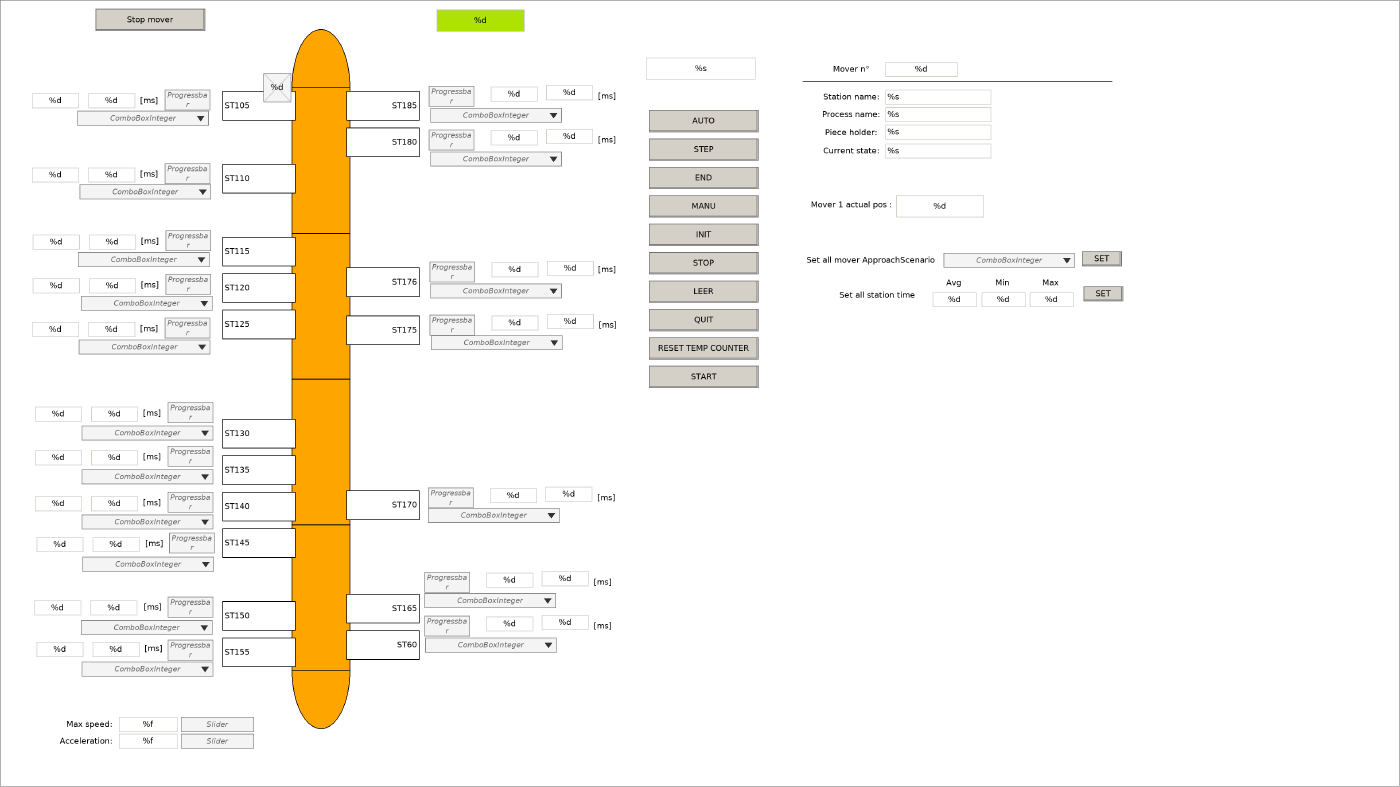
VISUALIZATION VISU_main  // 1920x1080
    Ellipse (400,840 80x160)
    Rectangle (400,720 80x200)
    Rectangle (400,520 80x200)
    Rectangle (400,320 80x200)
    Ellipse (400,40 80x160)
    Rectangle (400,120 80x200)
    Button (890,151 150x30), "AUTO", colour toggle: HMI.btArMain[0].on, input disabled if: HMI.btArMain[0].disable
        tap HMI.btArMain[0].button
    Button (890,190 150x30), "STEP", colour toggle: HMI.btArMain[1].on, input disabled if: HMI.btArMain[1].disable
        tap HMI.btArMain[1].button
    Button (890,229 150x30), "END", colour toggle: HMI.btArMain[2].on, input disabled if: HMI.btArMain[2].disable
        tap HMI.btArMain[2].button
    Button (890,307 150x30), "INIT", colour toggle: HMI.btArMain[4].on, input disabled if: HMI.btArMain[4].disable
        tap HMI.btArMain[4].button
    Button (890,346 150x30), "STOP", colour toggle: HMI.btArMain[5].disable, input disabled if: HMI.btArMain[5].disable
        tap HMI.btArMain[5].button
    Button (890,385 150x30), "LEER", colour toggle: HMI.btArMain[6].disable, input disabled if: HMI.btArMain[6].disable
        tap HMI.btArMain[6].button
    Button (890,424 150x30), "QUIT", colour toggle: HMI.btArMain[7].disable, input disabled if: HMI.btArMain[7].disable
        tap HMI.btArMain[7].button
    Button (890,463 150x30), "RESET TEMP COUNTER", colour toggle: HMI.btArMain[8].disable, input disabled if: HMI.btArMain[8].disable
        tap HMI.btArMain[8].button
    Button (890,268 150x30), "MANU", colour toggle: HMI.btArMain[3].on, input disabled if: HMI.btArMain[3].disable
        tap HMI.btArMain[3].button
    Textfield (886,79 150x30), "%s", text variable: _14_STATE.sStateDbg
    Button (890,502 150x30), "START", colour toggle: HMI.btArMain[9].disable, input disabled if: HMI.btArMain[9].disable
        tap HMI.btArMain[9].button
    Rectangle (475,175 100x40), "ST180", colour toggle: NOT PRG.st180_aut.xMoverPathFree
    Rectangle (475,367 100x40), "ST176", colour toggle: NOT PRG.st176_aut.xMoverPathFree
    Rectangle (475,433 100x40), "ST175", colour toggle: NOT PRG.st170_aut.xMoverPathFree
    Rectangle (475,673 100x40), "ST170", colour toggle: NOT PRG.st170_aut.xMoverPathFree
    Rectangle (475,815 100x40), "ST165", colour toggle: NOT PRG.st165_aut.xMoverPathFree
    Rectangle (475,865 100x40), "ST60", colour toggle: NOT PRG.st160_aut.xMoverPathFree
    Rectangle (305,875 100x40), "ST155", colour toggle: NOT PRG.st155_aut.xMoverPathFree
    Rectangle (475,125 100x40), "ST185", colour toggle: NOT PRG.st185_aut.xMoverPathFree
    Progressbar (588,178 62x28), variable: SIMU.iCompletionHMI[17]
    Progressbar (589,359 62x28), variable: SIMU.iCompletionHMI[16]
    Progressbar (589,432 62x28), variable: SIMU.iCompletionHMI[15]
    Progressbar (587,669 62x28), variable: SIMU.iCompletionHMI[14]
    Progressbar (582,785 62x28), variable: SIMU.iCompletionHMI[13]
    Progressbar (582,845 62x28), variable: SIMU.iCompletionHMI[12]
    Progressbar (230,878 62x28), variable: SIMU.iCompletionHMI[11]
    Progressbar (588,118 62x28), variable: SIMU.iCompletionHMI[18]
    Textfield (749,177 64x20), "%d", text variable: PERS.iStationTimeDef2[17]
        OnMouseDown: write the text variable via Default
    Label (805,177 55x30), "[ms]"
    Textfield (750,358 64x20), "%d", text variable: PERS.iStationTimeDef2[16]
        OnMouseDown: write the text variable via Default
    Label (805,355 55x30), "[ms]"
    Textfield (750,431 64x20), "%d", text variable: PERS.iStationTimeDef2[15]
        OnMouseDown: write the text variable via Default
    Label (806,431 55x30), "[ms]"
    Textfield (748,668 64x20), "%d", text variable: PERS.iStationTimeDef2[14]
        OnMouseDown: write the text variable via Default
    Label (804,668 55x30), "[ms]"
    Textfield (743,784 64x20), "%d", text variable: PERS.iStationTimeDef2[13]
        OnMouseDown: write the text variable via Default
    Label (799,784 55x30), "[ms]"
    Textfield (743,844 64x20), "%d", text variable: PERS.iStationTimeDef2[12]
        OnMouseDown: write the text variable via Default
    Label (799,844 55x30), "[ms]"
    Textfield (127,881 64x20), "%d", text variable: PERS.iStationTimeDef2[11]
        OnMouseDown: write the text variable via Default
    Label (183,875 55x30), "[ms]"
    Textfield (749,117 64x20), "%d", text variable: PERS.iStationTimeDef2[18]
        OnMouseDown: write the text variable via Default
    Label (805,117 55x30), "[ms]"
    Textfield (1229,268 120x30), "%d", text variable: MAIN.MoverMan._MoverList[1]._MoverAxis._CurrentPos
        OnMouseDown: write the text variable via Default
    Label (1080,266 146x30), "Mover 1 actual pos :"
    Textfield (599,13 120x30), "%d", text variable: PERS.iRecipeCurrent
        OnMouseDown: write the text variable via Default
    ComboBoxInteger (590,148 180x20), variable: MAIN.MoverMan._StationList[18]._ApproachScenario
    ComboBoxInteger (590,208 180x20), variable: MAIN.MoverMan._StationList[17]._ApproachScenario
    ComboBoxInteger (590,389 180x20), variable: MAIN.MoverMan._StationList[16]._ApproachScenario
    ComboBoxInteger (591,460 180x20), variable: MAIN.MoverMan._StationList[15]._ApproachScenario
    ComboBoxInteger (587,697 180x20), variable: MAIN.MoverMan._StationList[14]._ApproachScenario
    ComboBoxInteger (582,814 180x20), variable: MAIN.MoverMan._StationList[13]._ApproachScenario
    ComboBoxInteger (583,875 180x20), variable: MAIN.MoverMan._StationList[12]._ApproachScenario
    ComboBoxInteger (112,908 180x20), variable: MAIN.MoverMan._StationList[11]._ApproachScenario
    Rectangle (305,825 100x40), "ST150", colour toggle: NOT PRG.st150_aut.xMoverPathFree
    Progressbar (230,819 62x28), variable: SIMU.iCompletionHMI[10]
    Textfield (124,824 64x20), "%d", text variable: PERS.iStationTimeDef2[10]
        OnMouseDown: write the text variable via Default
    Label (182,818 55x30), "[ms]"
    ComboBoxInteger (111,851 180x20), variable: MAIN.MoverMan._StationList[10]._ApproachScenario
    Textfield (127,737 64x20), "%d", text variable: PERS.iStationTimeDef2[9]
        OnMouseDown: write the text variable via Default
    Label (184,731 55x30), "[ms]"
    Rectangle (305,725 100x40), "ST145", colour toggle: NOT PRG.st105_aut.xMoverPathFree
    Progressbar (232,731 62x28), variable: SIMU.iCompletionHMI[9]
    ComboBoxInteger (113,764 180x20), variable: MAIN.MoverMan._StationList[9]._ApproachScenario
    Textfield (125,681 64x20), "%d", text variable: PERS.iStationTimeDef2[8]
        OnMouseDown: write the text variable via Default
    Label (181,675 55x30), "[ms]"
    Rectangle (305,675 100x40), "ST140", colour toggle: NOT PRG.st140_aut.xMoverPathFree
    Progressbar (230,675 62x28), variable: SIMU.iCompletionHMI[8]
    ComboBoxInteger (112,706 180x20), variable: MAIN.MoverMan._StationList[8]._ApproachScenario
    Textfield (125,618 64x20), "%d", text variable: PERS.iStationTimeDef2[7]
        OnMouseDown: write the text variable via Default
    Label (181,612 55x30), "[ms]"
    Rectangle (305,625 100x40), "ST135", colour toggle: NOT PRG.st135_aut.xMoverPathFree
    Progressbar (230,612 62x28), variable: SIMU.iCompletionHMI[7]
    ComboBoxInteger (112,644 180x20), variable: MAIN.MoverMan._StationList[7]._ApproachScenario
    Textfield (125,558 64x20), "%d", text variable: PERS.iStationTimeDef2[6]
        OnMouseDown: write the text variable via Default
    Label (181,552 55x30), "[ms]"
    Rectangle (305,575 100x40), "ST130", colour toggle: NOT PRG.st130_aut.xMoverPathFree
    Progressbar (230,552 62x28), variable: SIMU.iCompletionHMI[6]
    ComboBoxInteger (112,584 180x20), variable: MAIN.MoverMan._StationList[6]._ApproachScenario
    Textfield (121,442 64x20), "%d", text variable: PERS.iStationTimeDef2[5]
        OnMouseDown: write the text variable via Default
    Label (177,436 55x30), "[ms]"
    Rectangle (305,425 100x40), "ST125", colour toggle: NOT PRG.st125_aut.xMoverPathFree
    Progressbar (226,436 62x28), variable: SIMU.iCompletionHMI[5]
    ComboBoxInteger (108,466 180x20), variable: MAIN.MoverMan._StationList[5]._ApproachScenario
    Textfield (122,382 64x20), "%d", text variable: PERS.iStationTimeDef2[4]
        OnMouseDown: write the text variable via Default
    Label (178,376 55x30), "[ms]"
    Rectangle (305,375 100x40), "ST120", colour toggle: NOT PRG.st120_aut.xMoverPathFree
    Progressbar (227,376 62x28), variable: SIMU.iCompletionHMI[4]
    ComboBoxInteger (111,406 180x20), variable: MAIN.MoverMan._StationList[4]._ApproachScenario
    Textfield (122,322 64x20), "%d", text variable: PERS.iStationTimeDef2[3]
        OnMouseDown: write the text variable via Default
    Label (178,316 55x30), "[ms]"
    Rectangle (305,325 100x40), "ST115", colour toggle: NOT PRG.st115_aut.xMoverPathFree
    Progressbar (227,316 62x28), variable: SIMU.iCompletionHMI[3]
    ComboBoxInteger (107,346 180x20), variable: MAIN.MoverMan._StationList[3]._ApproachScenario
    Textfield (121,230 64x20), "%d", text variable: PERS.iStationTimeDef2[2]
        OnMouseDown: write the text variable via Default
    Label (177,224 55x30), "[ms]"
    Rectangle (305,225 100x40), "ST110", colour toggle: NOT PRG.st110_aut.xMoverPathFree
    Progressbar (226,224 62x28), variable: SIMU.iCompletionHMI[2]
    ComboBoxInteger (109,253 180x20), variable: MAIN.MoverMan._StationList[2]._ApproachScenario
    Rectangle (305,125 100x40), "ST105", colour toggle: NOT PRG.st105_aut.xMoverPathFree
    Progressbar (226,123 62x28), variable: SIMU.iCompletionHMI[1]
    Textfield (121,128 64x20), "%d", text variable: PERS.iStationTimeDef2[1]
        OnMouseDown: write the text variable via Edit
    Label (177,123 55x30), "[ms]"
    ComboBoxInteger (106,152 180x20), variable: MAIN.MoverMan._StationList[1]._ApproachScenario
    ComboBoxInteger (1294,347 180x20), variable: MAIN.MoverMan.HMI_Scenario
    Label (1098,342 187x30), "Set all mover ApproachScenario"
    Button (1484,345 54x20), "SET"
        OnMouseDown: execute { MAIN.MoverMan.SetAllScenario(); }
    Label (1132,390 126x30), "Set all station time"
    Textfield (1279,401 60x20), "%d", text variable: MAIN.MoverMan.HMI_TimeAvg
        OnMouseDown: write the text variable via Default
    Label (1280,377 56x22), "Avg"
    Textfield (1346,401 60x20), "%d", text variable: MAIN.MoverMan.HMI_TimeMin
        OnMouseDown: write the text variable via Default
    Label (1347,377 56x22), "Min"
    Textfield (1412,401 60x20), "%d", text variable: MAIN.MoverMan.HMI_TimeMax
        OnMouseDown: write the text variable via Default
    Label (1413,377 56x22), "Max"
    Button (1486,393 54x20), "SET"
        OnMouseDown: execute { MAIN.MoverMan.SetAllTimers(ADR(PERS.iStationTimeDef1), 0); MAIN.MoverMan.SetAllTimers(ADR(PERS.iStationTimeDef2), 500); }
    Button (131,12 150x30), "Stop mover", colour toggle: MAIN.MoverMan.HMI_xStopMover
        toggle MAIN.MoverMan.HMI_xStopMover
    Label (1118,80 99x30), "Mover n°"
    Line (1101,111) (1525,111)
    Label (1118,118 99x30), "Station name:"
    Label (1118,142 99x30), "Process name:"
    Label (1118,167 99x30), "Piece holder:"
    Label (1118,192 99x30), "Current state:"
    Textfield (1214,85 99x20), "%d", text variable: MAIN.MoverMan.HMI_iSelMover
        OnMouseDown: write the text variable via Default
    Textfield (1214,123 145x20), "%s", text variable: MAIN.MoverMan._MoverList[MAIN.MoverMan.HMI_iSelMover].Station.ToString()
    Textfield (1214,147 145x20), "%s", text variable: MAIN.MoverMan._MoverList[MAIN.MoverMan.HMI_iSelMover].Station.Process.ToString()
    Textfield (1214,171 145x20), "%s"
    Textfield (1214,197 145x20), "%s", text variable: TO_STRING(MAIN.MoverMan._MoverList[MAIN.MoverMan.HMI_iSelMover]._State)
    Image (361,100 38x40), "%d", text variable: MAIN.MoverMan._MoverList[1]._ID, colour toggle: MAIN.MoverMan._SimuMoverList[1]._xStuck, invisible if: MAIN.MoverMan._MoverList[1]._MoverAxis._iID>CONST.MOVER_NUMBER, image: Custom.MoverSimu_final
        p3560616238: MAIN.MoverMan._MoverList[1]._MoverAxis.outSimuCurrentPos.x
        p2738717112: MAIN.MoverMan._MoverList[1]._MoverAxis.outSimuCurrentPos.y
        p2858320360: -MAIN.MoverMan._MoverList[1]._MoverAxis.outSimuCurrentRot
    Image (361,100 38x40), "%d", text variable: MAIN.MoverMan._MoverList[2]._ID, colour toggle: MAIN.MoverMan._SimuMoverList[2]._xStuck, invisible if: MAIN.MoverMan._MoverList[2]._MoverAxis._iID>CONST.MOVER_NUMBER, image: Custom.MoverSimu_final
        p3560616238: MAIN.MoverMan._MoverList[2]._MoverAxis.outSimuCurrentPos.x
        p2738717112: MAIN.MoverMan._MoverList[2]._MoverAxis.outSimuCurrentPos.y
        p2858320360: -MAIN.MoverMan._MoverList[2]._MoverAxis.outSimuCurrentRot
    Image (361,100 38x40), "%d", text variable: MAIN.MoverMan._MoverList[3]._ID, colour toggle: MAIN.MoverMan._SimuMoverList[3]._xStuck, invisible if: MAIN.MoverMan._MoverList[3]._MoverAxis._iID>CONST.MOVER_NUMBER, image: Custom.MoverSimu_final
        p3560616238: MAIN.MoverMan._MoverList[3]._MoverAxis.outSimuCurrentPos.x
        p2738717112: MAIN.MoverMan._MoverList[3]._MoverAxis.outSimuCurrentPos.y
        p2858320360: -MAIN.MoverMan._MoverList[3]._MoverAxis.outSimuCurrentRot
    Image (361,100 38x40), "%d", text variable: MAIN.MoverMan._MoverList[4]._ID, colour toggle: MAIN.MoverMan._SimuMoverList[4]._xStuck, invisible if: MAIN.MoverMan._MoverList[4]._MoverAxis._iID>CONST.MOVER_NUMBER, image: Custom.MoverSimu_final
        p3560616238: MAIN.MoverMan._MoverList[4]._MoverAxis.outSimuCurrentPos.x
        p2738717112: MAIN.MoverMan._MoverList[4]._MoverAxis.outSimuCurrentPos.y
        p2858320360: -MAIN.MoverMan._MoverList[4]._MoverAxis.outSimuCurrentRot
    Image (361,100 38x40), "%d", text variable: MAIN.MoverMan._MoverList[5]._ID, colour toggle: MAIN.MoverMan._SimuMoverList[5]._xStuck, invisible if: MAIN.MoverMan._MoverList[5]._MoverAxis._iID>CONST.MOVER_NUMBER, image: Custom.MoverSimu_final
        p3560616238: MAIN.MoverMan._MoverList[5]._MoverAxis.outSimuCurrentPos.x
        p2738717112: MAIN.MoverMan._MoverList[5]._MoverAxis.outSimuCurrentPos.y
        p2858320360: -MAIN.MoverMan._MoverList[5]._MoverAxis.outSimuCurrentRot
    Image (361,100 38x40), "%d", text variable: MAIN.MoverMan._MoverList[6]._ID, colour toggle: MAIN.MoverMan._SimuMoverList[6]._xStuck, invisible if: MAIN.MoverMan._MoverList[6]._MoverAxis._iID>CONST.MOVER_NUMBER, image: Custom.MoverSimu_final
        p3560616238: MAIN.MoverMan._MoverList[6]._MoverAxis.outSimuCurrentPos.x
        p2738717112: MAIN.MoverMan._MoverList[6]._MoverAxis.outSimuCurrentPos.y
        p2858320360: -MAIN.MoverMan._MoverList[6]._MoverAxis.outSimuCurrentRot
    Image (361,100 38x40), "%d", text variable: MAIN.MoverMan._MoverList[7]._ID, colour toggle: MAIN.MoverMan._SimuMoverList[7]._xStuck, invisible if: MAIN.MoverMan._MoverList[7]._MoverAxis._iID>CONST.MOVER_NUMBER, image: Custom.MoverSimu_final
        p3560616238: MAIN.MoverMan._MoverList[7]._MoverAxis.outSimuCurrentPos.x
        p2738717112: MAIN.MoverMan._MoverList[7]._MoverAxis.outSimuCurrentPos.y
        p2858320360: -MAIN.MoverMan._MoverList[7]._MoverAxis.outSimuCurrentRot
    Image (361,100 38x40), "%d", text variable: MAIN.MoverMan._MoverList[8]._ID, colour toggle: MAIN.MoverMan._SimuMoverList[8]._xStuck, invisible if: MAIN.MoverMan._MoverList[8]._MoverAxis._iID>CONST.MOVER_NUMBER, image: Custom.MoverSimu_final
        p3560616238: MAIN.MoverMan._MoverList[8]._MoverAxis.outSimuCurrentPos.x
        p2738717112: MAIN.MoverMan._MoverList[8]._MoverAxis.outSimuCurrentPos.y
        p2858320360: -MAIN.MoverMan._MoverList[8]._MoverAxis.outSimuCurrentRot
    Image (361,100 38x40), "%d", text variable: MAIN.MoverMan._MoverList[9]._ID, colour toggle: MAIN.MoverMan._SimuMoverList[9]._xStuck, invisible if: MAIN.MoverMan._MoverList[9]._MoverAxis._iID>CONST.MOVER_NUMBER, image: Custom.MoverSimu_final
        p3560616238: MAIN.MoverMan._MoverList[9]._MoverAxis.outSimuCurrentPos.x
        p2738717112: MAIN.MoverMan._MoverList[9]._MoverAxis.outSimuCurrentPos.y
        p2858320360: -MAIN.MoverMan._MoverList[9]._MoverAxis.outSimuCurrentRot
    Image (361,100 38x40), "%d", text variable: MAIN.MoverMan._MoverList[10]._ID, colour toggle: MAIN.MoverMan._SimuMoverList[10]._xStuck, invisible if: MAIN.MoverMan._MoverList[10]._MoverAxis._iID>CONST.MOVER_NUMBER, image: Custom.MoverSimu_final
        p3560616238: MAIN.MoverMan._MoverList[10]._MoverAxis.outSimuCurrentPos.x
        p2738717112: MAIN.MoverMan._MoverList[10]._MoverAxis.outSimuCurrentPos.y
        p2858320360: -MAIN.MoverMan._MoverList[10]._MoverAxis.outSimuCurrentRot
    Image (361,100 38x40), "%d", text variable: MAIN.MoverMan._MoverList[11]._ID, colour toggle: MAIN.MoverMan._SimuMoverList[11]._xStuck, invisible if: MAIN.MoverMan._MoverList[11]._MoverAxis._iID>CONST.MOVER_NUMBER, image: Custom.MoverSimu_final
        p3560616238: MAIN.MoverMan._MoverList[11]._MoverAxis.outSimuCurrentPos.x
        p2738717112: MAIN.MoverMan._MoverList[11]._MoverAxis.outSimuCurrentPos.y
        p2858320360: -MAIN.MoverMan._MoverList[11]._MoverAxis.outSimuCurrentRot
    Image (361,100 38x40), "%d", text variable: MAIN.MoverMan._MoverList[12]._ID, colour toggle: MAIN.MoverMan._SimuMoverList[12]._xStuck, invisible if: MAIN.MoverMan._MoverList[12]._MoverAxis._iID>CONST.MOVER_NUMBER, image: Custom.MoverSimu_final
        p3560616238: MAIN.MoverMan._MoverList[12]._MoverAxis.outSimuCurrentPos.x
        p2738717112: MAIN.MoverMan._MoverList[12]._MoverAxis.outSimuCurrentPos.y
        p2858320360: -MAIN.MoverMan._MoverList[12]._MoverAxis.outSimuCurrentRot
    Image (361,100 38x40), "%d", text variable: MAIN.MoverMan._MoverList[13]._ID, colour toggle: MAIN.MoverMan._SimuMoverList[13]._xStuck, invisible if: MAIN.MoverMan._MoverList[13]._MoverAxis._iID>CONST.MOVER_NUMBER, image: Custom.MoverSimu_final
        p3560616238: MAIN.MoverMan._MoverList[13]._MoverAxis.outSimuCurrentPos.x
        p2738717112: MAIN.MoverMan._MoverList[13]._MoverAxis.outSimuCurrentPos.y
        p2858320360: -MAIN.MoverMan._MoverList[13]._MoverAxis.outSimuCurrentRot
    Image (361,100 38x40), "%d", text variable: MAIN.MoverMan._MoverList[14]._ID, colour toggle: MAIN.MoverMan._SimuMoverList[14]._xStuck, invisible if: MAIN.MoverMan._MoverList[14]._MoverAxis._iID>CONST.MOVER_NUMBER, image: Custom.MoverSimu_final
        p3560616238: MAIN.MoverMan._MoverList[14]._MoverAxis.outSimuCurrentPos.x
        p2738717112: MAIN.MoverMan._MoverList[14]._MoverAxis.outSimuCurrentPos.y
        p2858320360: -MAIN.MoverMan._MoverList[14]._MoverAxis.outSimuCurrentRot
    Image (361,100 38x40), "%d", text variable: MAIN.MoverMan._MoverList[15]._ID, colour toggle: MAIN.MoverMan._SimuMoverList[15]._xStuck, invisible if: MAIN.MoverMan._MoverList[15]._MoverAxis._iID>CONST.MOVER_NUMBER, image: Custom.MoverSimu_final
        p3560616238: MAIN.MoverMan._MoverList[15]._MoverAxis.outSimuCurrentPos.x
        p2738717112: MAIN.MoverMan._MoverList[15]._MoverAxis.outSimuCurrentPos.y
        p2858320360: -MAIN.MoverMan._MoverList[15]._MoverAxis.outSimuCurrentRot
    Image (361,100 38x40), "%d", text variable: MAIN.MoverMan._MoverList[16]._ID, colour toggle: MAIN.MoverMan._SimuMoverList[16]._xStuck, invisible if: MAIN.MoverMan._MoverList[16]._MoverAxis._iID>CONST.MOVER_NUMBER, image: Custom.MoverSimu_final
        p3560616238: MAIN.MoverMan._MoverList[16]._MoverAxis.outSimuCurrentPos.x
        p2738717112: MAIN.MoverMan._MoverList[16]._MoverAxis.outSimuCurrentPos.y
        p2858320360: -MAIN.MoverMan._MoverList[16]._MoverAxis.outSimuCurrentRot
    Image (361,100 38x40), "%d", text variable: MAIN.MoverMan._MoverList[17]._ID, colour toggle: MAIN.MoverMan._SimuMoverList[17]._xStuck, invisible if: MAIN.MoverMan._MoverList[17]._MoverAxis._iID>CONST.MOVER_NUMBER, image: Custom.MoverSimu_final
        p3560616238: MAIN.MoverMan._MoverList[17]._MoverAxis.outSimuCurrentPos.x
        p2738717112: MAIN.MoverMan._MoverList[17]._MoverAxis.outSimuCurrentPos.y
        p2858320360: -MAIN.MoverMan._MoverList[17]._MoverAxis.outSimuCurrentRot
    Image (361,100 38x40), "%d", text variable: MAIN.MoverMan._MoverList[18]._ID, colour toggle: MAIN.MoverMan._SimuMoverList[18]._xStuck, invisible if: MAIN.MoverMan._MoverList[18]._MoverAxis._iID>CONST.MOVER_NUMBER, image: Custom.MoverSimu_final
        p3560616238: MAIN.MoverMan._MoverList[18]._MoverAxis.outSimuCurrentPos.x
        p2738717112: MAIN.MoverMan._MoverList[18]._MoverAxis.outSimuCurrentPos.y
        p2858320360: -MAIN.MoverMan._MoverList[18]._MoverAxis.outSimuCurrentRot
    Image (361,100 38x40), "%d", text variable: MAIN.MoverMan._MoverList[19]._ID, colour toggle: MAIN.MoverMan._SimuMoverList[19]._xStuck, invisible if: MAIN.MoverMan._MoverList[19]._MoverAxis._iID>CONST.MOVER_NUMBER, image: Custom.MoverSimu_final
        p3560616238: MAIN.MoverMan._MoverList[19]._MoverAxis.outSimuCurrentPos.x
        p2738717112: MAIN.MoverMan._MoverList[19]._MoverAxis.outSimuCurrentPos.y
        p2858320360: -MAIN.MoverMan._MoverList[19]._MoverAxis.outSimuCurrentRot
    Textfield (163,984 80x20), "%f", text variable: SIMU.lrSpeedMover
    Textfield (163,1007 80x20), "%f", text variable: SIMU.lrAccelMover
    Label (57,984 100x20), "Max speed:"
    Label (57,1007 100x20), "Acceleration:"
    Slider (248,984 100x20), variable: SIMU.lrSpeedMover, scale 1..50
    Slider (248,1007 100x20), variable: SIMU.lrAccelMoverSlider, scale 0.1..1
    Textfield (50,881 64x20), "%d", text variable: PERS.iStationTimeDef1[11]
        OnMouseDown: write the text variable via Default
    Textfield (47,824 64x20), "%d", text variable: PERS.iStationTimeDef1[10]
        OnMouseDown: write the text variable via Default
    Textfield (50,737 64x20), "%d", text variable: PERS.iStationTimeDef1[9]
        OnMouseDown: write the text variable via Default
    Textfield (48,681 64x20), "%d", text variable: PERS.iStationTimeDef1[8]
        OnMouseDown: write the text variable via Default
    Textfield (48,618 64x20), "%d", text variable: PERS.iStationTimeDef1[7]
        OnMouseDown: write the text variable via Default
    Textfield (48,558 64x20), "%d", text variable: PERS.iStationTimeDef1[6]
        OnMouseDown: write the text variable via Default
    Textfield (44,442 64x20), "%d", text variable: PERS.iStationTimeDef1[5]
        OnMouseDown: write the text variable via Default
    Textfield (45,382 64x20), "%d", text variable: PERS.iStationTimeDef1[4]
        OnMouseDown: write the text variable via Default
    Textfield (45,322 64x20), "%d", text variable: PERS.iStationTimeDef1[3]
        OnMouseDown: write the text variable via Default
    Textfield (44,230 64x20), "%d", text variable: PERS.iStationTimeDef1[2]
        OnMouseDown: write the text variable via Default
    Textfield (44,128 64x20), "%d", text variable: PERS.iStationTimeDef1[1]
        OnMouseDown: write the text variable via Edit
    Textfield (673,179 64x20), "%d", text variable: PERS.iStationTimeDef1[17]
        OnMouseDown: write the text variable via Default
    Textfield (674,360 64x20), "%d", text variable: PERS.iStationTimeDef1[16]
        OnMouseDown: write the text variable via Default
    Textfield (674,433 64x20), "%d", text variable: PERS.iStationTimeDef1[15]
        OnMouseDown: write the text variable via Default
    Textfield (672,670 64x20), "%d", text variable: PERS.iStationTimeDef1[14]
        OnMouseDown: write the text variable via Default
    Textfield (667,786 64x20), "%d", text variable: PERS.iStationTimeDef1[13]
        OnMouseDown: write the text variable via Default
    Textfield (667,846 64x20), "%d", text variable: PERS.iStationTimeDef1[12]
        OnMouseDown: write the text variable via Default
    Textfield (673,119 64x20), "%d", text variable: PERS.iStationTimeDef1[18]
        OnMouseDown: write the text variable via Default
END_VISUALIZATION

(* stored: Version 1.1.0.1, ProductVersion 3.1.4024.12
   Visu VISU_main: Id {d72905fe-72a6-4ef2-acdb-6547139e7766} *)
